{attribute 'TcGenerated'}
{attribute 'no-analysis'}
{attribute 'linkalways'}
// This function has been automatically generated from the project information.
VAR_GLOBAL CONSTANT
	{attribute 'const_non_replaced'}
	stLibVersion_GDT_Utilities_Library : ST_LibVersion := (iMajor := 0, iMinor := 1, iBuild := 0, iRevision := 0, nFlags := 0, sVersion := '0.1.0.0');
END_VAR

(* stored: Version 1.1.0.1, ProductVersion 3.1.4024.9
   GVL Global_Version: Id {6207c0e6-370a-47cf-b15c-03f145ee68f5} *)
